(* PLC project SafeLOGIC-1, BrAutomation SafeDESIGNER  4.3.4.4 *)
(* stored: companyURL http://www.br-automation.com, creationDateTime Thu Jun 24 15:41:11 2021 *)

PROGRAM Main
  VAR  (* added by the conversion: wires and edge detectors of the diagram *)
    _SAFEBOOL_TO_BOOL6_OUT : BOOL;
  END_VAR

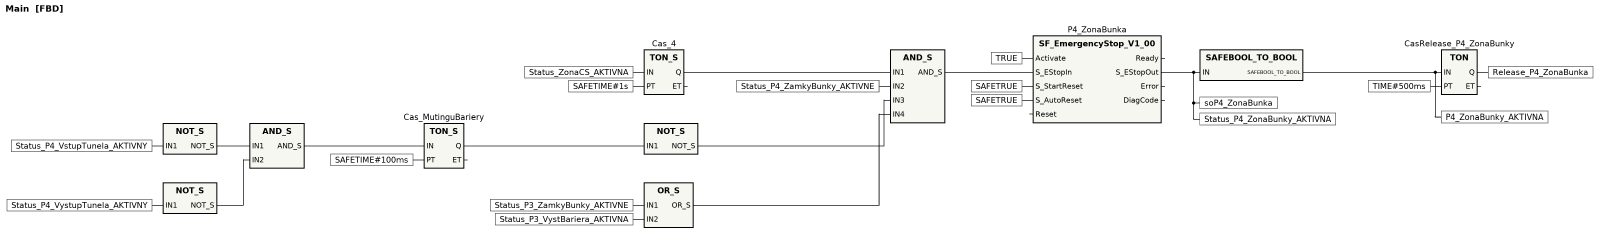
(* FBD diagram, written out as Structured Text *)
Cas_4(IN := Status_ZonaCS_AKTIVNA, PT := SAFETIME#1s);
Cas_MutinguBariery(IN := AND_S(NOT_S(Status_P4_VstupTunela_AKTIVNY), NOT_S(Status_P4_VystupTunela_AKTIVNY)), PT := SAFETIME#100ms);
P4_ZonaBunka(Activate := TRUE, S_EStopIn := AND_S(Cas_4.Q, Status_P4_ZamkyBunky_AKTIVNE, NOT_S(Cas_MutinguBariery.Q), OR_S(Status_P3_ZamkyBunky_AKTIVNE, Status_P3_VystBariera_AKTIVNA)), S_StartReset := SAFETRUE, S_AutoReset := SAFETRUE);
Status_P4_ZonaBunky_AKTIVNA := P4_ZonaBunka.S_EStopOut;
soP4_ZonaBunka := P4_ZonaBunka.S_EStopOut;
_SAFEBOOL_TO_BOOL6_OUT := SAFEBOOL_TO_BOOL(P4_ZonaBunka.S_EStopOut);
P4_ZonaBunky_AKTIVNA := _SAFEBOOL_TO_BOOL6_OUT;
CasRelease_P4_ZonaBunky(IN := _SAFEBOOL_TO_BOOL6_OUT, PT := TIME#500ms);
Release_P4_ZonaBunka := CasRelease_P4_ZonaBunky.Q;
END_PROGRAM
